// TIA Portal V19 export
FUNCTION "PRESTERILIZING" : Void   // FC40, STL
TITLE = PRESTERILIZING ASEPTIC TANK
{ S7_Optimized_Access := 'TRUE' }
NAME : TNKSTERI
VERSION : 0.0
// Comment
// stored: AutoNumber false
BEGIN

NETWORK
TITLE = PRESTERILIZING ASEPTIC TANK
      AN    "S0 PRESTERILIZING";
      R     "S1 PRESTERILIZING";
      R     "S2 PRESTERILIZING";
      R     "S3 PRESTERILIZING";
      R     "S4 PRESTERILIZING";
      R     "S5 PRESTERILIZING";
      R     "S6 PRESTERILIZING";
      R     "S7 PRESTERILIZING";
      BEC;
      A     "S1 PRESTERILIZING";
      JC    M001;
      S     "MY0545";
      S     "MY0148";
      R     "MY0103";
      S     "MY0104";
      S     "MY0136";
      R     "MY0137";
      S     "MY0135";
      S     "MY0143";
      R     "MY0111";
      R     "MY0109";
      R     "MY0108";
      R     "MY0124";
      R     "MY0144";
      S     "MY0112";
      R     "MY0113";
      S     "MY0118";
      R     "MY0147";
//    S     "MY01.14"
      R     "MY0101";
//    R     "MM01.30"
      R     "AutoPT0167/IP0149";
      R     "ManPT0167/IP0149";
      R     "PULSE 01.18 PRESTERILI";
      R     "SPIN 01.30 PRESTERILI";
      R     "TEST TEMPS. PRESTERILI";
      R     "TEST BARRIERS";
      R     "TANK STERILE";

      R     "StopFillers_UHT_Rec";
//;
      S     "MY0904";
      S     "MY0907";
      S     "IF_Device".V_09_30.IO.V._IO.IN.Activate;
      A     "Y0904S";  //check valve energised
      A     "Y0907S";  //check valve energised
      A     "IF_Device".V_09_30.IO.V._IO.OUT.ValveOpened;
      JCN   NW1E;

      R     "MY0901";
      R     "MY0905";
      R     "MY0906";
      R     "MY0912";
      A     "Y0905R";  //check valve de-energised
      A     "Y0906R";  //check valve de-energised
      A     "Y0912R";  //check valve de-energised
      JCN   NW1E;

      S     "S1 PRESTERILIZING";
//;
NW1E: BEU;
M001: NOP   0;

NETWORK
TITLE = Q 9.5; Output modul 1 Channel 13
      A     "S2 PRESTERILIZING";
      JC    c001;
      L     "MeasuredValues".TT0176REAL;  // "DB-ANALOG INPUT".TT0176MEAS
      L     "Setpoints".CloseY0113;  //"DB SETPOINTS".CloseY0113   // 95,0 C
      <R;
      BEC;
      R     "MY0118";
      S     "PULSE 01.18 PRESTERILI";
      S     "SPIN 01.30 PRESTERILI";
      S     "S2 PRESTERILIZING";
      BEU;
c001: NOP   0;

NETWORK
TITLE = START TIMER 14
      A     "S3 PRESTERILIZING";
      JC    c002;
      A(;
      L     "MeasuredValues".TT0176REAL;  //"DB-ANALOG INPUT".TT0176MEAS
      L     "Setpoints".TT0176StartSterileTime;  //"DB SETPOINTS".TT0176StartSterileTime
      <R;
      );
      BEC;
      A(;
      L     "MeasuredValues".TT0160REAL;  //"DB-ANALOG INPUT".TT0160MEAS
      L     "Setpoints".TT0160StartSterileTime;  //"DB SETPOINTS".TT0160StartSterileTime
      <R;
      );
      BEC;
      A(;
      L     "MeasuredValues".TT0163REAL;  // "DB-ANALOG INPUT".TT0163MEAS
      L     "Setpoints".TT0163StartSterileTime;  //"DB SETPOINTS".TT0163StartSterileTime
      <R;
      );
      BEC;
      A(;
      L     "MeasuredValues".TT0178REAL;  // "DB-ANALOG INPUT".TT0178MEAS
      L     "Setpoints".TT0178StartSterileTime;  //"DB SETPOINTS".TT0178StartSterileTime
      <R;
      );
      BEC;
      A(;
      L     "MeasuredValues".TT0951REAL;  // "DB-ANALOG INPUT".TT0951MEAS
      L     "Setpoints_Hamba".TT0951StartSterileTime;  //"DB SETPOINTS".TT0951StartSterileTime
      <R;
      );
      BEC;
      A(;
      L     "PG_Devices".TTX0940.Value;
      L     "Setpoints_Polygon".TT0940_Low_SIP;
      <R;
      );
      BEC;
      S     "TIM14";
      S     "TEST TEMPS. PRESTERILI";
      S     "M_Barrier_Sterlising";
      S     "S3 PRESTERILIZING";
      BEU;
c002: NOP   0;

NETWORK
TITLE = Q 8.2; Output modul 1 Channel 2
      A     "S4 PRESTERILIZING";
      JC    c003;
      A     "T 14 STERILE TIME";  //
//     A     M     50.0                  //step on


      BEC;
      R     "MY0104";
      S     "MY0137";
      S     "MY0109";
      R     "MY0545";
      R     "MY0112";
      S     "MY0147";
      R     "PULSE 01.18 PRESTERILI";
      R     "MY0118";
      R     "TEST TEMPS. PRESTERILI";
      S     "TEST BARRIERS";
      S     "TIM15";
      R     "MY0143";
      R     "SPIN 01.30 PRESTERILI";
//     R     "MM01.30"
      S     "TANK STERILE";
      S     "TEST FILLING PRESSURE";

//;
      R     "MY0904";
      S     "MY0906";
      S     "MY0901";
      A     "Y0904R";  //check valve de-energised
      A     "Y0906S";  //check valve energised
      JCN   NW4E;

      S     "S4 PRESTERILIZING";
//;
NW4E: BEU;
c003: NOP   0;

NETWORK
TITLE = Q 8.3; Output modul 1 Channel 3
      A     "S5 PRESTERILIZING";
      JC    c004;
      A     "T 15 COOLING TIME";
      JC    M002;
      R     "MY0109";
      S     "S5 PRESTERILIZING";
      BEU;
M002: L     "MeasuredValues".PT0167REAL;  //"DB-ANALOG INPUT".PT0167MeasPressure
      L     "Setpoints".PT0167StopCooling;  //"DB SETPOINTS".PT0167StopCooling
      >R;
      JC    M003;
      R     "MY0109";
      BEU;
M003: L     "MeasuredValues".PT0167REAL;  //"DB-ANALOG INPUT".PT0167MeasPressure
      L     "Setpoints".PT0167RestartCooling;  //"DB SETPOINTS".PT0167RestartCooling
      >R;
      JC    M004;
      BEU;
M004: S     "MY0109";
      AN    "AutoPT0167/IP0149";
      JC    M005;
      BEU;
M005: L     "MeasuredValues".PT0167REAL;  //"DB-ANALOG INPUT".PT0167MeasPressure
      L     1.8;
      >R;
      BEC;
      S     "MY0111";
      L     "Setpoints".PT0167SpInCooling;  //"DB SETPOINTS".PT0167SpInCooling
      T     "STP_PT0167/IP0149_50".PT0167SpSTP;
      S     "AutoPT0167/IP0149";
      L     1200;
      T     "STP_PT0167/IP0149_50".IP0149OutSTP;
      BEU;
c004: NOP   0;

NETWORK
TITLE = Q 8.5; Output modul 1 Channel 5
// Comment
      A     "S6 PRESTERILIZING";
      JC    c005;
      L     "MeasuredValues".PT0167REAL;  //"DB-ANALOG INPUT".PT0167MeasPressure
      L     "Setpoints".StartBlowOutMinPressure;  //"DB SETPOINTS".StartBlowOutMinPressure
      <R;
      BEC;
      S     "MY0112";
      S     "MY0118";
      R     "MY0147";
      S     "TIM16";
      S     "S6 PRESTERILIZING";
      BEU;
c005: NOP   0;

NETWORK
TITLE = Q 8.5; Output modul 1 Channel 5
      A     "S7 PRESTERILIZING";
      JC    c006;
      A     "T 16 BLOW OUT COND";
      BEC;
      R     "MY0112";
      R     "MY0118";
      S     "MY0147";
      L     "Setpoints".PT0167SpProduction;  //"DB SETPOINTS".PT0167SpProduction
      T     "STP_PT0167/IP0149_50".PT0167SpSTP;
      S     "ProcessAndPbAlarms"."A"[39];  //A39_TankReadyforProd// tank ready for production
      S     "S7 PRESTERILIZING";
//;
      S     "M_Barrier_Sterile";
      R     "M_Barrier_Sterlising";
//;
      BEU;
c006: NOP   0;

NETWORK
TITLE = 
// Comment
      S     "S0 PRODUCTION TANK";
      R     "S0 PRESTERILIZING";
      S     "LEDAssignment".K3_LIGHT;  //"LIGHT_K3_PRESTE."
      S     "LEDAssignment".K3_FLASH;  //"FLASH_K3_PRESTE."
      BEU;
END_FUNCTION
